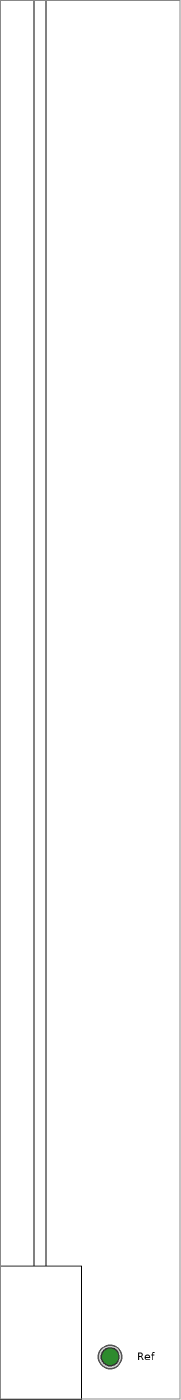
VISUALIZATION Lift_Axis  // 189x1460
VAR_IN_OUT
	Position : REAL;
	RefSensor : BOOL;
END_VAR
    Rectangle (35,0 13x1460)
    Lamp1 (100,1400 30x30), variable: RefSensor, style: Lamp-Lamp1-Green
    Rectangle (0,1320 85x140)
        p2738717112: - (1320.0 / 100.0 * Position)
    Label (140,1400 49x30), "Ref"
END_VISUALIZATION

(* stored: Version 1.1.0.1
   Visu Lift_Axis: Id {21aa2dc7-7e08-4a3b-8abf-bbb625916ca0} *)
